TYPE ST_INPUTS_StaticConv:
STRUCT
	
	Mode:     	E_DeviceMode;
	Command:    E_DeviceState;

END_STRUCT
END_TYPE

(* stored: Version 1.1.0.1, ProductVersion 3.1.4024.12
   DUT ST_INPUTS_StaticConv: Id {2d4527d7-6b6b-4787-805a-1027439f47b6} *)
